DATA_BLOCK "MyDB"
NON_RETAIN

"U_Status"

BEGIN

critical := false;

END_DATA_BLOCK